TYPE ST_StorageDock :
STRUCT	
	sName				: STRING;
	nId					: INT;
	refStorage			: REFERENCE TO FB_Storage;
	posOrigin			: ST_Coordinate;
	bTeached			: BOOL;
	
END_STRUCT
END_TYPE

(* stored: Version 1.1.0.1
   DUT ST_StorageDock: Id {2b900ed2-445b-4410-8051-93a71088bbbe} *)
